(* IEC 61131-3 sources: POMIRTS_lab3/AS/Library/AsSMTP, 3 files *)

(* ---- AsSMTP.typ ---- *)
(********************************************************************
 * COPYRIGHT -- Bernecker + Rainer
 ********************************************************************
 * Library: AsSMTP
 * File: AsSMTP.typ
 * Author: B+R
 ********************************************************************
 * Data types of library AsSMTP
 ********************************************************************)

TYPE
    smtpATTACHMENT_typ	: STRUCT		(*attachments*)
		type			: UDINT;		(*type of attachment (file, module or memory area)*)
		pData			: UDINT;		(*pointer to the data (depends on attachment type: filename, modulename or memory address)*)
		length			: UDINT;		(*length of memory (only for memory attachments)*)
		pName			: UDINT;		(*name of attachment (optional, default: filename, modulename or mematt_<# of attachment>)*)
	END_STRUCT;
END_TYPE

(* ---- AsSMTP.fun ---- *)
(********************************************************************
 * COPYRIGHT -- Bernecker + Rainer
 ********************************************************************
 * Library: AsSMTP
 * File: AsSMTP.fun
 * Author: B+R
 ********************************************************************
 * Functions and function blocks of library AsSMTP
 ********************************************************************)

FUNCTION_BLOCK SmtpSend					(*sends email; asynchronous execution*)
	VAR_INPUT
		enable			: BOOL;			(*enables execution*)
		pHost			: UDINT;		(*pointer to the ip address of mail server*)
		pUser			: UDINT;		(*pointer to the user name for authentication*)
		pPassword		: UDINT;		(*pointer to the password for authentication*)
		pSender			: UDINT;		(*pointer to the name of sender*)
		pReceiver		: UDINT;		(*pointer to the ip addresses of receiver*)
		pSubject		: UDINT;		(*pointer to the subject string*)
		pText			: UDINT;		(*pointer to the text string*)
		pDomain			: UDINT;		(*pointer to the sender domain*)
		pAttachment		: UDINT;		(*pointer to the attachment structure field*)
		pSecurity		: UDINT;		(*reserved for future use*)
		timeout			: UDINT;		(*response timeout for connection establishment with smtp server*)
		port			: UINT;			(*port of mail server*)
		attcnt			: USINT;		(*number of attachments*)
	END_VAR

	VAR_OUTPUT
		status			: UINT;			(*execution status: ERR_OK, ERR_FUB_ENABLE_FALSE, ERR_FUB_BUSY, 0xXXXX = see help*)
	END_VAR

	VAR
        i_state			: UINT;			(*internal variable*)
		i_result		: UINT;			(*internal variable*)
        i_tmp			: UDINT;		(*internal variable*)
	END_VAR
END_FUNCTION_BLOCK

(* ---- AsSMTP.var ---- *)
(********************************************************************
 * COPYRIGHT -- Bernecker + Rainer
 ********************************************************************
 * Library: AsSMTP
 * File: AsSMTP.var
 * Author: B+R
 ********************************************************************
 * Local variables of library AsSMTP
 ********************************************************************)

VAR CONSTANT

	smtpERR_PARAMETER					: UINT := 32700;	(*invalid parameter, check parameter*)
	smtpERR_SOCKET_CREATE				: UINT := 32701;	(*create socket failed*)
	smtpERR_SOCKET_CONNECT				: UINT := 32702;	(*connect socket failed*)
	smtpERR_RESPONSE_TIMEOUT			: UINT := 32703;	(*server response timeout*)
	smtpERR_RESPONSE_UNEXPECTED			: UINT := 32704;	(*unexpected response*)
	smtpERR_AUTHENTICATION_METHOD		: UINT := 32705;	(*no supported authentication method*)
	smtpERR_AUTHENTICATION_FAILED		: UINT := 32706;	(*authentication failed*)
	smtpERR_ATTACHMENT_INVALID			: UINT := 32707;	(*invalid attachment*)

	smtpERR_SYSTEM						: UINT := 32749;	(*system error*)

	smtpATT_TYPE_FILE					: USINT := 1;		(*attachment type file*)
	smtpATT_TYPE_DATMOD					: USINT := 2;		(*attachment type datamodule*)
	smtpATT_TYPE_MEMORY					: USINT := 3;		(*attachment type memory area*)
END_VAR
